VISUALIZATION vLock  // 2x2
END_VISUALIZATION

(* stored: Version 1.1.0.1, ProductVersion 3.1.4024.15
   Visu vLock: Id {4db6f3cc-2e69-4529-8143-2e8d8aee5f0b} *)
